TYPE ST_System_HOWW_Zustand :
STRUCT
	Betrieb_Anford			: BOOL;
	Betrieb_Soll				: BOOL;
	Betrieb					: BOOL;

	Netze_Anford				: ST_Zustand_Netze_Anford;

	Freigabe					: BOOL;
	Freigabe_Deakt			: BOOL;
	Freigabe_Code			: WORD;

	Stoerung					: BOOL;
	Stoerung_Code			: WORD;

	Warnung					: BOOL;
	Warnung_Code			: WORD;

	Status					: SINT;
	Status_Vorl_Regelventil		: BOOL;
	Status_Vorl_Pumpe		: BOOL;
	Status_Nachl_Regelventil	: BOOL;
	Status_Nachl_Pumpe		: BOOL;

	Quittierung				: BOOL;

	Netz_WW_Anford			: ST_Zustand_Netz_Anford; (* Philipp *)

END_STRUCT
END_TYPE

(* stored: Version 1.1.0.1, ProductVersion 3.1.4024.9
   DUT ST_System_HOWW_Zustand: Id {e87a1927-7c7c-49ba-865c-f9b0f4651ffa} *)
